(* LS Electric XG5000 project: 05_Practice2_TON_TOF *)
(* PLC LSPLC *)
(* module base 0 slot 0: 입력 모듈:XGI-D21A (DC 24V 입력, 8점 (전류소스/싱크입력)) *)
(* module base 0 slot 1: 출력 모듈:XGQ-RY1A (릴레이 출력, 8점 (2A용, 단독 COM.)) *)

PROGRAM NewProgram (* task: 스캔 프로그램 *)
VAR
    램프 AT %QX0.1.0 : BOOL;
    스위치 AT %IX0.0.0 : BOOL;
    시간입력 : TIME := T#0s;
    타이머1 : TON;
    타이머2 : TOF;
END_VAR

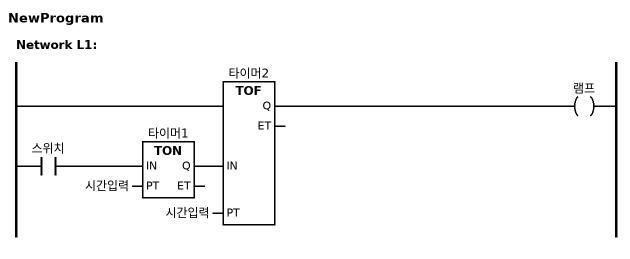
(* Rung L1 *)
타이머1(IN := 스위치, PT := 시간입력);
타이머2(IN := 타이머1.Q, PT := 시간입력);
램프 := 타이머2.Q;
END_PROGRAM